# EPICS substitutions: vacuum/MAIN_TRUNK/vacApp/Db/l417_agilent4uhv.substitutions
# Agilent4UHV substitutions file

file db/agilent4uhv.db
{
     pattern {LOCA,			DEV,			PORT,		ADDR,	TIMEOUT}
     		{HL4,			VL417_1,		4uhv_1,		0,		0.2}
     		{HL4,			VL417_2,		4uhv_2,		0,		0.2}
}

file db/agilent4uhv_alias.db
{
     pattern {LOCA,			DEV,			SUB1,				SUB2,				SUB3,					SUB4,				PORT,		ADDR,	TIMEOUT}
     		 {HL4,			VL417_1,		IP01:L417_Acc601,		IP02:L417_Acc602,		IP03:L417_Acc603,			IP04:L417_Acc604,		4uhv_1,		0,		0.2}
		 {HL4,			VL417_2,		IP05:L417_Acc605,		IP06:L417_Wave601,	IP07:L417_Kly601,			IP08:Empty,			4uhv_2,		0,		0.2}
}
